INTERFACE I_ActuatorStartStop EXTENDS I_ActuatorBase

{attribute 'monitoring' := 'call'}
PROPERTY public isStarted : BOOL
GET
END_GET
END_PROPERTY

{attribute 'monitoring' := 'call'}
PROPERTY public isStopped : BOOL
GET
END_GET
END_PROPERTY

METHOD public start : BOOL
VAR_INPUT
END_VAR
END_METHOD

METHOD public stop : BOOL
VAR_INPUT
END_VAR
END_METHOD

END_INTERFACE

(* stored: Version 1.1.0.1, ProductVersion 3.1.4024.3
   Itf I_ActuatorStartStop: Id {2f4c6c16-e270-4a9f-b923-7191b52f6674}
   Property isStarted: Id {038ef8c5-3402-4f4b-8523-6bf22a2e3740}
   Get Get: Id {59dfe0b0-675a-4791-a01d-9f6d96880725}
   Property isStopped: Id {b9382c80-d2db-4f38-bdfc-fa90ed67707b}
   Get Get: Id {28a90c06-16c5-4982-8cb4-f65d9e296d85}
   Method start: Id {7344032b-0c29-438c-bad4-e8c235e48be1}
   Method stop: Id {86f38d89-3dcb-45ac-9193-b7287b2c500e} *)
